{attribute 'qualified_only'}
TYPE ENUM_Coating_States :
(
	Unknown := 0,
    Coating1 := 1,
    Coating2 := 2
);
END_TYPE

(* stored: Version 1.1.0.1, ProductVersion 3.1.4022.18
   DUT ENUM_Coating_States: Id {118e1a24-82d2-4598-99ea-540bbe0bbd1a} *)
